{attribute addProperty BoxType "EL5101-0011-0016"}
{attribute addProperty Id "StartTimeNextLatchAT %I*ULINT648"}
{attribute addProperty CRC "1335715474"}
{attribute addProperty SizeInBites "64"}
{attribute addProperty SizeInBytes "8"}
TYPE ENC_NextSync1Time_4F9D6692 :
STRUCT
	{attribute addProperty Name "StartTimeNextLatch"}
	StartTimeNextLatch AT %I* : ULINT;
END_STRUCT
END_TYPE

(* stored: Version 1.2.0.0, ProductVersion 3.1.4024.9
   DUT ENC_NextSync1Time_4F9D6692: Id {11be7192-f19a-4427-b72b-a1cdbc915358} *)
